TYPE SBoolExpressionSpec :
STRUCT
	Operator: EBoolOperation;
	
	LeftType: EExpressionType;
	LeftIdx: UINT;
	
	RightType: EExpressionType;
	RightIdx: UINT;
END_STRUCT
END_TYPE

(* stored: Version 1.1.0.1, ProductVersion 3.1.4024.9
   DUT SBoolExpressionSpec: Id {556423ce-123e-4fa9-8a4f-80d9e1a13e8a} *)
